{attribute 'GeneratedUsingTerminal: EL2912-0000-0016'}
{attribute addProperty BoxType "EL2912-0000-0016"}
{attribute addProperty Id "OutputsOutputs_8B1C946D2"}
{attribute addProperty CRC "1834791005"}
{attribute addProperty Size "2"}
TYPE Module_2_FSOUT_6D5CB05D :
STRUCT
	{attribute addProperty Name "Outputs"}
	Outputs  : Outputs_8B1C946D;
END_STRUCT
END_TYPE

(* stored: Version 1.2.0.0, ProductVersion 3.1.4024.9
   DUT Module_2_FSOUT_6D5CB05D: Id {16455f93-8f7a-4c04-8d39-51de0eea91c2} *)
